(* Logix 5000 project; controller PLC_Safety vendor 1 type 14 code 148 rev 37.11; software revision 37.00; part 3 of 3 *)
(* tags used below, declared in another part *)
   Auto_OK : BOOL;
   Fanuc_Enable : BOOL;
   Gate_1 : DCI_STOP;
   Gate_1_State : BOOL;
   Gate_2 : DCI_STOP;
   Gate_2_State : BOOL;
   GuardLock_OK : BOOL;
   LightCurtain : DCI_STOP;
   LightCurtain_OK : BOOL;
   LightCurtain_State : BOOL;
   Manual_OK : BOOL;
   OSF_Reset_G1 : BOOL;
   OSF_Reset_G2 : BOOL;
   OSF_Reset_P1 : BOOL;
   OSF_Reset_P2 : BOOL;
   Reset_G1 : BOOL;
   Reset_G2 : BOOL;
   Reset_P1 : BOOL;
   Reset_P2 : BOOL;
   Safety_Mat_OK : BOOL;
   SafetyScanner1 : DCI_STOP;
   SafetyScanner1_OK : BOOL;
   SafetyScanner1_State : BOOL;
   SafetyScanner2 : DCI_STOP;
   SafetyScanner2_OK : BOOL;
   SafetyScanner2_State : BOOL;
   Servo_Drive_1_Enable : BOOL;
   Servo_Drive_1_Status_OK : BOOL;
   Servo_Drive_2_Enable : BOOL;
   Servo_Drive_2_Status_OK : BOOL;
   true : BOOL;
   VFD_1_Enable : BOOL;
   VFD_1_Status_OK : BOOL;
   VFD_2_Enable : BOOL;
   VFD_2_Status_OK : BOOL;
   E_Stop_OK : BOOL;
   Gate_1_Open_SFTY : ALIAS FOR Point_IO_Gabinete_1:6:I.Pt07Data;   // Push Button Gate 1 Open
   Gate_1_Reset_SFTY : ALIAS FOR Point_IO_Gabinete_1:6:I.Pt06Data;   // Push Button Gate 1 Reset
   Gate_2_Open_SFTY : BOOL;   // Push Button Gate 2 Open
   Gate_2_Reset_SFTY : BOOL;   // Push Button Gate 2 Reset
   Manual_SFTY : BOOL;
   Process_1_Reset_SFTY : BOOL;   // Push Button Process 1 Reset
   Process_2_Reset_SFTY : ALIAS FOR Point_IO_Gabinete_2:6:I.Pt06Data;   // Push Button Process 2 Reset
   Reset_General : BOOL;
   Safety_OK : BOOL;
(* SafetyProgram, continued *)

ROUTINE R02_Light_Curtain   (* ladder *)
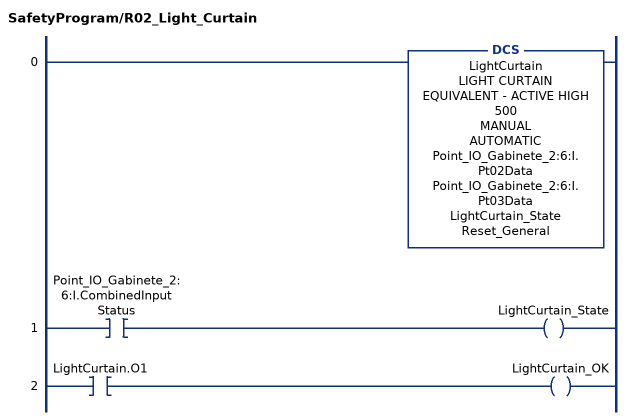
   0: DCS(LightCurtain,LIGHT CURTAIN,EQUIVALENT - ACTIVE HIGH,500,MANUAL,AUTOMATIC,Point_IO_Gabinete_2:6:I.Pt02Data,Point_IO_Gabinete_2:6:I.Pt03Data,LightCurtain_State,Reset_General);
   1: XIC(Point_IO_Gabinete_2:6:I.CombinedInputStatus)OTE(LightCurtain_State);
   2: XIC(LightCurtain.O1)OTE(LightCurtain_OK);
END_ROUTINE

ROUTINE R03_Safety_Mat   (* ladder *)
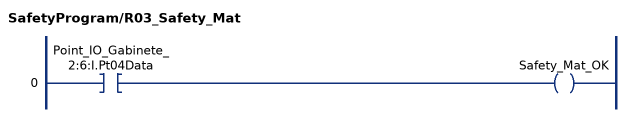
   0: XIC(Point_IO_Gabinete_2:6:I.Pt04Data)OTE(Safety_Mat_OK);
END_ROUTINE

ROUTINE R04_SafetyScanner   (* ladder *)
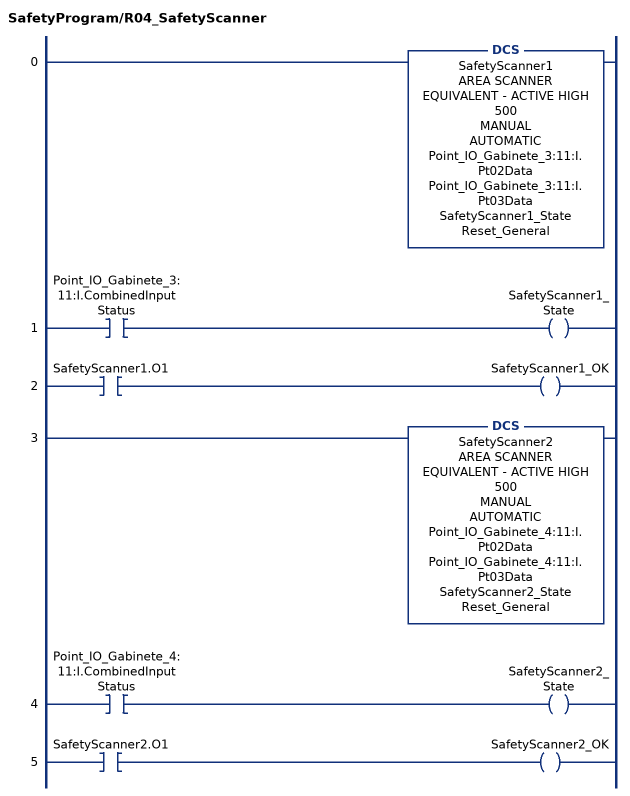
   0: DCS(SafetyScanner1,AREA SCANNER,EQUIVALENT - ACTIVE HIGH,500,MANUAL,AUTOMATIC,Point_IO_Gabinete_3:11:I.Pt02Data,Point_IO_Gabinete_3:11:I.Pt03Data,SafetyScanner1_State,Reset_General);
   1: XIC(Point_IO_Gabinete_3:11:I.CombinedInputStatus)OTE(SafetyScanner1_State);
   2: XIC(SafetyScanner1.O1)OTE(SafetyScanner1_OK);
   3: DCS(SafetyScanner2,AREA SCANNER,EQUIVALENT - ACTIVE HIGH,500,MANUAL,AUTOMATIC,Point_IO_Gabinete_4:11:I.Pt02Data,Point_IO_Gabinete_4:11:I.Pt03Data,SafetyScanner2_State,Reset_General);
   4: XIC(Point_IO_Gabinete_4:11:I.CombinedInputStatus)OTE(SafetyScanner2_State);
   5: XIC(SafetyScanner2.O1)OTE(SafetyScanner2_OK);
END_ROUTINE

ROUTINE R05_GuardLock   (* ladder *)
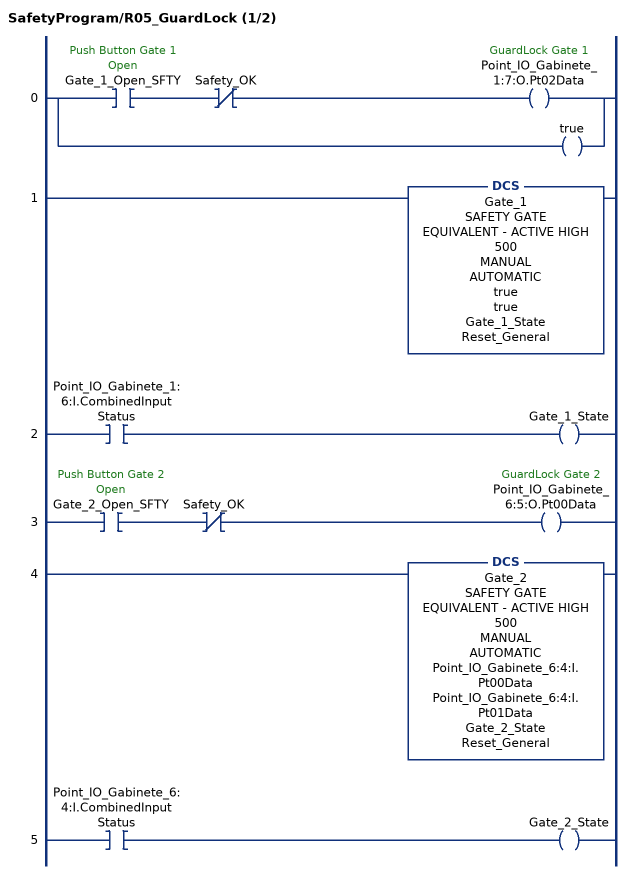
   0: [XIC(Gate_1_Open_SFTY) XIO(Safety_OK) OTE(Point_IO_Gabinete_1:7:O.Pt02Data) ,OTE(true) ];
   1: DCS(Gate_1,SAFETY GATE,EQUIVALENT - ACTIVE HIGH,500,MANUAL,AUTOMATIC,true,true,Gate_1_State,Reset_General);
   2: XIC(Point_IO_Gabinete_1:6:I.CombinedInputStatus)OTE(Gate_1_State);
   3: XIC(Gate_2_Open_SFTY)XIO(Safety_OK)OTE(Point_IO_Gabinete_6:5:O.Pt00Data);
   4: DCS(Gate_2,SAFETY GATE,EQUIVALENT - ACTIVE HIGH,500,MANUAL,AUTOMATIC,Point_IO_Gabinete_6:4:I.Pt00Data,Point_IO_Gabinete_6:4:I.Pt01Data,Gate_2_State,Reset_General);
   5: XIC(Point_IO_Gabinete_6:4:I.CombinedInputStatus)OTE(Gate_2_State);
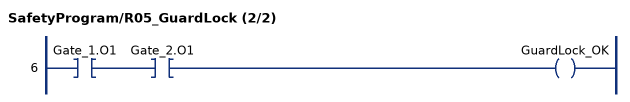
   6: XIC(Gate_1.O1)XIC(Gate_2.O1)OTE(GuardLock_OK);
END_ROUTINE

ROUTINE R06_Safety_OK   (* ladder *)
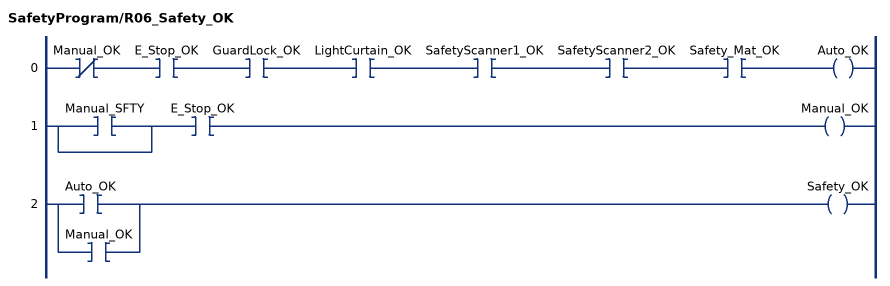
   0: XIO(Manual_OK)XIC(E_Stop_OK)XIC(GuardLock_OK)XIC(LightCurtain_OK)XIC(SafetyScanner1_OK)XIC(SafetyScanner2_OK)XIC(Safety_Mat_OK)OTE(Auto_OK);
   1: [XIC(Manual_SFTY) ,]XIC(E_Stop_OK)OTE(Manual_OK);
   2: [XIC(Auto_OK) ,XIC(Manual_OK) ]OTE(Safety_OK);
END_ROUTINE

ROUTINE R07_Reset   (* ladder *)
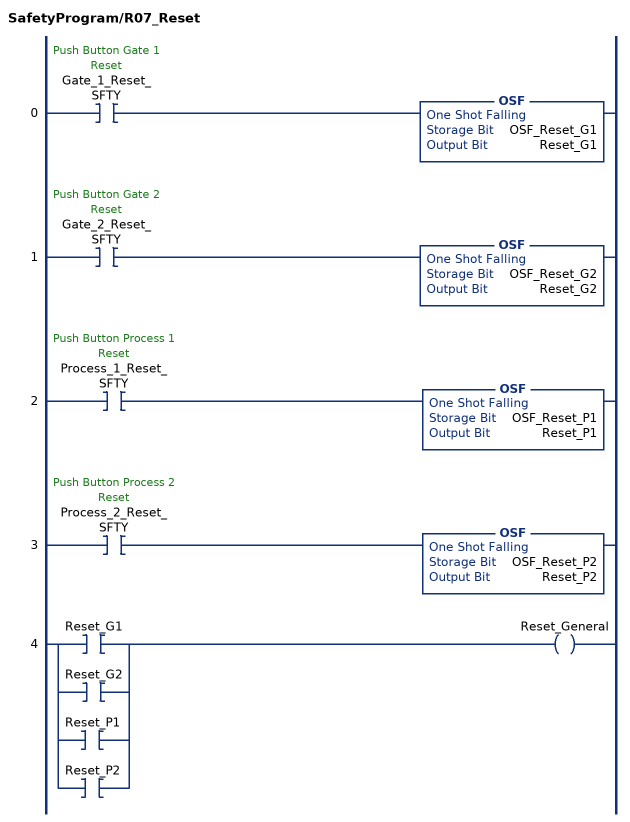
   0: XIC(Gate_1_Reset_SFTY)OSF(OSF_Reset_G1,Reset_G1);
   1: XIC(Gate_2_Reset_SFTY)OSF(OSF_Reset_G2,Reset_G2);
   2: XIC(Process_1_Reset_SFTY)OSF(OSF_Reset_P1,Reset_P1);
   3: XIC(Process_2_Reset_SFTY)OSF(OSF_Reset_P2,Reset_P2);
   4: [XIC(Reset_G1) ,XIC(Reset_G2) ,XIC(Reset_P1) ,XIC(Reset_P2) ]OTE(Reset_General);
END_ROUTINE

ROUTINE R08_Motor   (* ladder *)
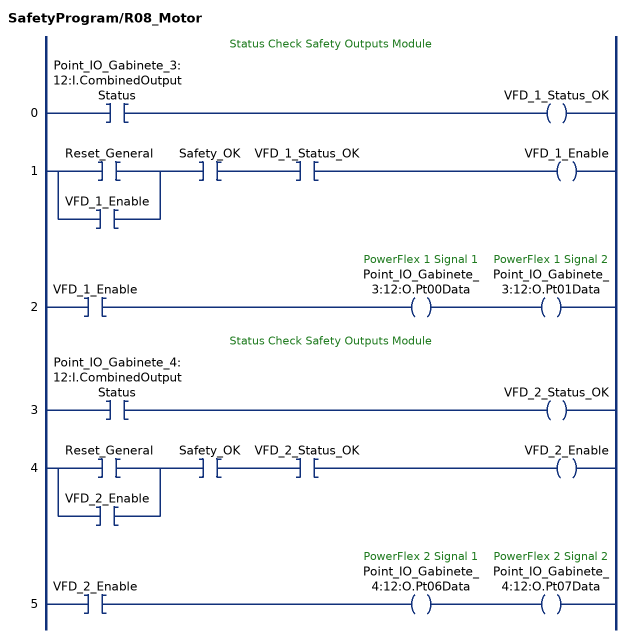
   // Status Check Safety Outputs Module
   0: XIC(Point_IO_Gabinete_3:12:I.CombinedOutputStatus)OTE(VFD_1_Status_OK);
   1: [XIC(Reset_General) ,XIC(VFD_1_Enable) ]XIC(Safety_OK)XIC(VFD_1_Status_OK)OTE(VFD_1_Enable);
   2: XIC(VFD_1_Enable)OTE(Point_IO_Gabinete_3:12:O.Pt00Data)OTE(Point_IO_Gabinete_3:12:O.Pt01Data);
   // Status Check Safety Outputs Module
   3: XIC(Point_IO_Gabinete_4:12:I.CombinedOutputStatus)OTE(VFD_2_Status_OK);
   4: [XIC(Reset_General) ,XIC(VFD_2_Enable) ]XIC(Safety_OK)XIC(VFD_2_Status_OK)OTE(VFD_2_Enable);
   5: XIC(VFD_2_Enable)OTE(Point_IO_Gabinete_4:12:O.Pt06Data)OTE(Point_IO_Gabinete_4:12:O.Pt07Data);
END_ROUTINE

ROUTINE R09_Servomotor   (* ladder *)
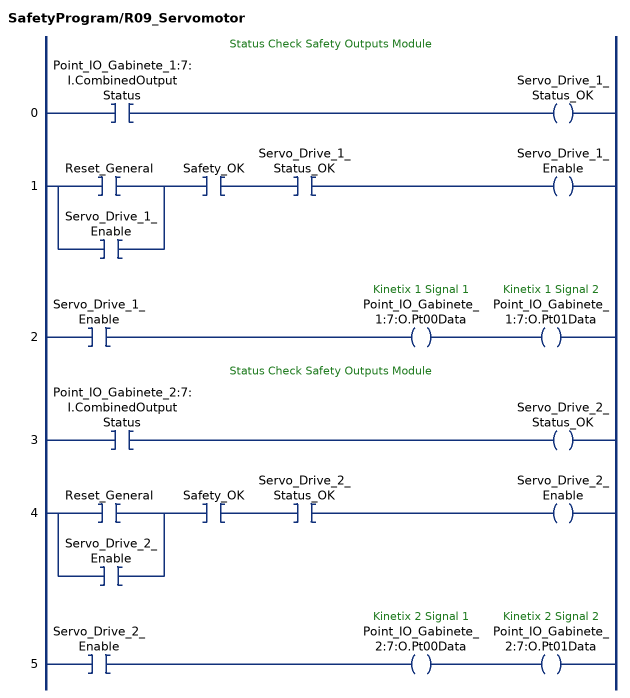
   // Status Check Safety Outputs Module
   0: XIC(Point_IO_Gabinete_1:7:I.CombinedOutputStatus)OTE(Servo_Drive_1_Status_OK);
   1: [XIC(Reset_General) ,XIC(Servo_Drive_1_Enable) ]XIC(Safety_OK)XIC(Servo_Drive_1_Status_OK)OTE(Servo_Drive_1_Enable);
   2: XIC(Servo_Drive_1_Enable)OTE(Point_IO_Gabinete_1:7:O.Pt00Data)OTE(Point_IO_Gabinete_1:7:O.Pt01Data);
   // Status Check Safety Outputs Module
   3: XIC(Point_IO_Gabinete_2:7:I.CombinedOutputStatus)OTE(Servo_Drive_2_Status_OK);
   4: [XIC(Reset_General) ,XIC(Servo_Drive_2_Enable) ]XIC(Safety_OK)XIC(Servo_Drive_2_Status_OK)OTE(Servo_Drive_2_Enable);
   5: XIC(Servo_Drive_2_Enable)OTE(Point_IO_Gabinete_2:7:O.Pt00Data)OTE(Point_IO_Gabinete_2:7:O.Pt01Data);
END_ROUTINE

ROUTINE R10_Fanuc_Safety   (* ladder *)
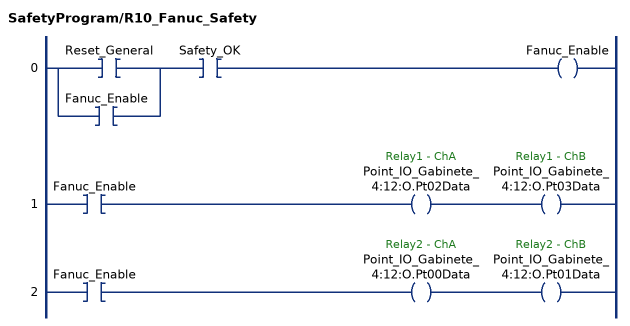
   0: [XIC(Reset_General) ,XIC(Fanuc_Enable) ]XIC(Safety_OK)OTE(Fanuc_Enable);
   1: XIC(Fanuc_Enable)OTE(Point_IO_Gabinete_4:12:O.Pt02Data)OTE(Point_IO_Gabinete_4:12:O.Pt03Data);
   2: XIC(Fanuc_Enable)OTE(Point_IO_Gabinete_4:12:O.Pt00Data)OTE(Point_IO_Gabinete_4:12:O.Pt01Data);
END_ROUTINE
END_PROGRAM
